// TwinCAT 3 PLC project Warehouse
// ProgramVersion: 3.1.4026.16
// CompilerDefines: VISU_USEPROPERTYINFO
// libraries:
//   Tc2_Standard, * (Beckhoff Automation GmbH)
//   Tc2_System, * (Beckhoff Automation GmbH)
//   VisuSymbols, 4.5.0.0 (System)
// project tree:
//   / GlobalTextList.TcGTLO (not stored), PlcTask.TcTTO
//   POUs/ FB_WarehouseStock.TcPOU, MAIN.TcPOU (not stored)
// real-time tasks:
//   TASK PlcTask: cycle T#10ms, priority 20, ADS port 350
//   TASK VISU_TASK: cycle T#200000us, priority 30, ADS port 351

CONFIGURATION Warehouse
    RESOURCE PLC ON TwinCAT3
        TASK PlcTask(INTERVAL := T#10ms, PRIORITY := 20);
        PROGRAM MAIN WITH PlcTask : MAIN;
    END_RESOURCE
END_CONFIGURATION

// ---- POUs/FB_WarehouseStock.TcPOU
FUNCTION_BLOCK FB_WarehouseStock
VAR_INPUT	
END_VAR
VAR_OUTPUT
END_VAR
VAR
	iXAxis:			INT;
	iYAxis:			INT;
	bStored:			BOOL;
	bRemoved:			BOOL;
	arrStockPosition:	ARRAY[1..7, 1..12] OF INT;
END_VAR

METHOD M_Remove : BOOL
VAR_INPUT
	iProdNumber: 		INT;
END_VAR
END_METHOD

METHOD M_Store : BOOL
VAR_INPUT
	iProdNumber: 		INT;
END_VAR
bStored := FALSE;

IF iProdNumber = 0 THEN
	RETURN;
END_IF

FOR iXAxis := 1 TO 7 BY 1 DO
	FOR iYAxis :=  1 TO 12 BY 1 DO
		IF arrStockPosition[iXAxis, iYAxis] = 0 THEN
			arrStockPosition[iXAxis, iYAxis] := iProdNumber;
			bStored := TRUE;
			EXIT;
		END_IF
		IF bStored = TRUE THEN
			RETURN;
		END_IF
	END_FOR
END_FOR
END_METHOD

END_FUNCTION_BLOCK
